//---------------------------------------------------------------------------------------------------------------
//
//  fb_Configuration
//
//  HAUD 2023.04.14
//  - base xml integration
//
//  HAUD 2026.04.10.
//  - now extending a base class
//
//  - cyclic OnChange wrapper for xml data 
//      - Ctrl/State
//        1. INIT
//        2. READ / WRITE
//
//  - read  ST_STATION_PARAMETER on demand
//  - write ST_STATION_PARAMETER on demand
//
//---------------------------------------------------------------------------------------------------------------
// This SOFTWARE is provided as an Example by THE PROVIDER "as is" and "with all faults." THE PROVIDER makes no 
// representations or warranties of any kind concerning the safety, suitability, lack of viruses, inaccuracies, 
// typographical errors, or other harmful components of this SOFTWARE. There are inherent dangers in the use of 
// any software, and you are solely responsible for determining whether this SOFTWARE is compatible with your 
// equipment and other software installed on your equipment. You are also solely responsible for the protection 
// of your equipment and backup of your data, and THE PROVIDER will not be liable for any damages you may suffer 
// in connection with using, modifying, or distributing this SOFTWARE.
//---------------------------------------------------------------------------------------------------------------
FUNCTION_BLOCK fb_Configuration EXTENDS fb_XmlBase
VAR
  _stCtrl               : REFERENCE TO ST_DATA_CTRL;
  _stState              : REFERENCE TO ST_DATA_STATE;

  _stConfiguration      : ST_Configuration;
  _pStationParameter    : POINTER TO ARRAY[1..MAX_STATION] OF ST_STATION_PARAMETER;
END_VAR
VAR CONSTANT
  FILE_ROOT             : STRING := 'CONFIG_XtsTransport_';
  X_PATH                : STRING := '/XtsTransport/config';
END_VAR

//---------------------------------------------------------------------------------------------------------------
//  check pointers from the outside
//---------------------------------------------------------------------------------------------------------------
IF NOT Check() THEN RETURN; END_IF
//---------------------------------------------------------------------------------------------------------------
// always build the internal data pointer
//  - as always: better safe than sorry
//  - leave this bit here, it doesn't cost much and safely addresses the data
//---------------------------------------------------------------------------------------------------------------
_pData                        := ADR    (_stConfiguration);
_nData                        := SIZEOF (_stConfiguration);
_sXpath                       := X_PATH;

// copy to local for debug
_eCmd                         := _stCtrl.Cmd;

// cyclic check for command change
// get state for cmd
IF (_eCmd <> _eCmdOld)
THEN
  // get matching sdtate for Ctrl.Cmd
  _eState                     := Cmd(_eCmd);
  _eCmdOld                    := _eCmd;
END_IF


CASE _eResult
OF
  E_PROGRESS.PROGRESS_INVALID:
    _stState.State            := E_DATA_STATE.NULL;

  E_PROGRESS.PROGRESS_ERROR:
    _stState.State            := _eState + E_PROGRESS.PROGRESS_ERROR;

  E_PROGRESS.PROGRESS_DONE:
    _stState.State            := _eState + E_PROGRESS.PROGRESS_DONE;

ELSE
  // work in progress
  // update progress for extern use
  _stState.State              := _eState + _eResult;

  CASE _eState
  OF
    E_DATA_STATE.INIT:
      _eResult   := _eInit    := CreateFolder(TRUE);

    E_DATA_STATE.READ:
      _eResult                := XmlRead(TRUE);
      IF (_eResult = E_PROGRESS.PROGRESS_DONE)
      THEN
        // copy the single ladies
        memcpy(_pStationParameter, ADR(_stConfiguration.XtsStationParameter), SIZEOF(_stConfiguration.XtsStationParameter));
      END_IF

    E_DATA_STATE.WRITE:
      _eResult                := XmlWrite(TRUE);
  ELSE
      _eResult                := E_PROGRESS.PROGRESS_INVALID;
  END_CASE
END_CASE

METHOD Check : BOOL
//-------------------------------------------------------------------------
IF NOT (__ISVALIDREF(_stCtrl))
THEN
  _eCheck               := E_DATA_CHECK.REFERENCE_CTRL_INVALID;
  RETURN;
END_IF
//-------------------------------------------------------------------------
IF NOT (__ISVALIDREF(_stState))
THEN
  _eCheck               := E_DATA_CHECK.REFERENCE_STATE_INVALID;
  RETURN;
END_IF
//-------------------------------------------------------------------------
IF NOT (_pStationParameter <> 0)
THEN
  _eCheck               := E_DATA_CHECK.POINTER_STATION_PARAMETER_INVALID;
  RETURN;
END_IF
//-------------------------------------------------------------------------
_eCheck                 := E_DATA_CHECK.DONE_CHECK;
Check                   := TRUE;
END_METHOD

METHOD PRIVATE Cmd : E_DATA_STATE
VAR_INPUT
  Ctrl      : E_DATA_CTRL;
END_VAR
VAR_INST
  _eState   : E_DATA_STATE;
END_VAR
IF NOT Check() THEN Cmd   := E_DATA_STATE.NULL;  RETURN; END_IF

CASE Ctrl
OF
  //---------------------------------------------------------------
  E_DATA_CTRL.INIT:
    _sName                := concat(FILE_ROOT, _sIdentity);
    _sName                := concat(_sName, '.xml');
    _sFilePath            := concat(_sDirectoryPath, _sName);

    _eInit                := E_PROGRESS.PROGRESS_INVALID;
    _eResult              := CreateFolder(FALSE);
    _eState               := E_DATA_STATE.INIT;
  //---------------------------------------------------------------
  E_DATA_CTRL.READ:
    _eResult              := XmlRead(FALSE);
    _eState               := E_DATA_STATE.READ;
  //---------------------------------------------------------------
  E_DATA_CTRL.WRITE:
    _stConfiguration.XtsStationParameter  := _pStationParameter^;

    _eResult              := XmlWrite(FALSE);
    _eState               := E_DATA_STATE.WRITE;
ELSE
  //---------------------------------------------------------------
    _eResult              := E_PROGRESS.PROGRESS_INVALID; 
    _eState               := E_DATA_STATE.NO_EXIST;
END_CASE

Cmd                       := _eState;
END_METHOD

PROPERTY Ctrl : REFERENCE to ST_DATA_CTRL
SET
_stCtrl ref= Ctrl;
END_SET
END_PROPERTY

PROPERTY Identity : OTCID
GET
Identity := _XpuIdentity;
END_GET
SET
_XpuIdentity  := Identity;
_sIdentity    := Tc2_Utilities.DWORD_TO_HEXSTR(_XpuIdentity,8,FALSE);
END_SET
END_PROPERTY

PROPERTY State : REFERENCE TO ST_DATA_STATE
SET
_stState ref= State;
END_SET
END_PROPERTY

PROPERTY StationParameter : pointer to ARRAY[1..MAX_STATION] OF ST_STATION_PARAMETER
SET
_pStationParameter := StationParameter;
END_SET
END_PROPERTY

END_FUNCTION_BLOCK

(* stored: Version 1.1.0.1
   POU fb_Configuration: Id {6e927e36-d027-4f8f-9bf1-0b498bb5e245}, SpecialFunc None
   Folder methods: Id {d27e853f-7731-4c6e-aec9-4fb7cfb5baab}
   Folder properties: Id {e378cae4-4de9-410b-9e79-b09f60ebb6d3}
   Method Check: Id {ebdfa161-0abf-405f-abc2-f1977b4c39ec}
   Method Cmd: Id {7ca34bc6-a226-44ae-8522-b796e20bd62b}
   Property Ctrl: Id {fca9a518-7ef7-4131-af16-8bdb0ef53e3e}
   Set Set: Id {a5af3173-ae57-4326-a8ab-8c58e82b06a0}
   Property Identity: Id {1ae4968c-043c-4c8e-bb1f-0cc8fb21f541}
   Get Get: Id {602817ad-235a-411a-992f-4c7ead53afcb}
   Set Set: Id {32fa3343-5135-463f-92ef-d1d9d0d3a5eb}
   Property State: Id {da92e3dd-9b27-4368-ba5f-069e8c78d5c9}
   Set Set: Id {df14fb62-84aa-49e4-a1b4-9bff583f18a2}
   Property StationParameter: Id {1f8da58c-9023-4b7b-a143-ca73e0aed437}
   Set Set: Id {854a5c78-30b6-48d8-ac61-3d6b06cf68de} *)
